{attribute 'qualified_only'}
{attribute 'strict'}
TYPE BuzzerType :
(
	ONCE := 0,
	CYCLE,
	OFF
);
END_TYPE

(* stored: Version 1.1.0.1, ProductVersion 3.1.4024.14
   DUT BuzzerType: Id {713c46c8-1c3d-46af-923c-8ac08de764ec} *)
